INTERFACE I_HomingCommand EXTENDS I_AxisCommand

END_INTERFACE

(* stored: Version 1.1.0.1, ProductVersion 3.1.4024.12
   Itf I_HomingCommand: Id {4aeda662-6f6c-4461-bfe4-562f47fed1ce} *)
